INTERFACE I_FallibleUdint


PROPERTY Error : BOOL
GET
END_GET
END_PROPERTY


PROPERTY Value : UDINT
GET
END_GET
END_PROPERTY

END_INTERFACE

(* stored: Version 1.1.0.1
   Itf I_FallibleUdint: Id {a1b2c3d4-0003-4001-8001-000000000021}
   Property Error: Id {a1b2c3d4-0003-4001-8001-000000000022}
   Get Get: Id {a1b2c3d4-0003-4001-8001-000000000023}
   Property Value: Id {a1b2c3d4-0003-4001-8001-000000000024}
   Get Get: Id {a1b2c3d4-0003-4001-8001-000000000025} *)
